LIN {X 0,Y 173.677,Z 475.724,A -85,B 0,C 180,E1 -30232.4,E2 -30232.4} C_VEL
LIN {X 0,Y 173.787,Z 475.712,A -85,B 0,C 180,E1 -30235.65,E2 -30235.65} C_VEL
LIN {X 0,Y 173.897,Z 476.638,A -85,B 0,C 180,E1 -30237.104,E2 -30237.104} C_VEL
LIN {X 0,Y 169.927,Z 506.64,A -85,B 0,C 180,E1 -30237.538,E2 -30237.538} C_VEL
LIN {X 0,Y 166.155,Z 523.912,A -85,B 0,C 180,E1 -30237.792,E2 -30237.792} C_VEL
LIN {X 0,Y 160.855,Z 540.987,A -85,B 0,C 180,E1 -30238.078,E2 -30238.078} C_VEL
LIN {X 0,Y 155.111,Z 555.302,A -85,B 0,C 180,E1 -30238.461,E2 -30238.461} C_VEL
LIN {X 0,Y 147.609,Z 570.627,A -85,B 0,C 180,E1 -30239.029,E2 -30239.029} C_VEL
LIN {X 0,Y 139.67,Z 584.169,A -85,B 0,C 180,E1 -30239.669,E2 -30239.669} C_VEL
LIN {X 0,Y 130.9,Z 596.782,A -85,B 0,C 180,E1 -30240.433,E2 -30240.433} C_VEL
LIN {X 0,Y 121.274,Z 608.767,A -85,B 0,C 180,E1 -30241.51,E2 -30241.51} C_VEL
LIN {X 0,Y 110.826,Z 620.073,A -85,B 0,C 180,E1 -30242.83,E2 -30242.83} C_VEL
LIN {X 0,Y 98.738,Z 631.287,A -85,B 0,C 180,E1 -30244.804,E2 -30244.804} C_VEL
LIN {X 0,Y 86.785,Z 640.843,A -85,B 0,C 180,E1 -30247.242,E2 -30247.242} C_VEL
LIN {X 0,Y 72.974,Z 650.367,A -85,B 0,C 180,E1 -30251.102,E2 -30251.102} C_VEL
LIN {X 0,Y 62.022,Z 656.96,A -85,B 0,C 180,E1 -30255.6,E2 -30255.6} C_VEL
LIN {X 0,Y 49.708,Z 663.438,A -85,B 0,C 180,E1 -30263.221,E2 -30263.221} C_VEL
LIN {X 0,Y 38.747,Z 668.721,A -85,B 0,C 180,E1 -30275.294,E2 -30275.294} C_VEL
LIN {X 0,Y 32.128,Z 671.865,A -85,B 0,C 180,E1 -30288.988,E2 -30288.988} C_VEL
LIN {X 0,Y 27.268,Z 675.138,A -85,B 0,C 180,E1 -30315.066,E2 -30315.066} C_VEL
LIN {X 0,Y 27.051,Z 676.337,A -85,B 0,C 180,E1 -30330.002,E2 -30330.002} C_VEL
LIN {X 0,Y 29.084,Z 677.949,A -85,B 0,C 180,E1 -30358.903,E2 -30358.903} C_VEL
LIN {X 0,Y 36.518,Z 678.543,A -85,B 0,C 180,E1 -30380.339,E2 -30380.339} C_VEL
LIN {X 0,Y 47.081,Z 678.294,A -85,B 0,C 180,E1 -30393.595,E2 -30393.595} C_VEL
LIN {X 0,Y 59.202,Z 677.038,A -85,B 0,C 180,E1 -30401.751,E2 -30401.751} C_VEL
LIN {X 0,Y 72.097,Z 674.944,A -85,B 0,C 180,E1 -30407.114,E2 -30407.114} C_VEL
LIN {X 0,Y 85.435,Z 671.806,A -85,B 0,C 180,E1 -30410.805,E2 -30410.805} C_VEL
LIN {X 0,Y 99.04,Z 667.758,A -85,B 0,C 180,E1 -30413.447,E2 -30413.447} C_VEL
LIN {X 0,Y 103.79,Z 666.021,A -85,B 0,C 180,E1 -30414.851,E2 -30414.851} C_VEL
LIN {X 0,Y 91.479,Z 669.945,A -85,B 0,C 180,E1 -30417.138,E2 -30417.138} C_VEL
LIN {X 0,Y 77.315,Z 673.389,A -85,B 0,C 180,E1 -30420.727,E2 -30420.727} C_VEL
LIN {X 0,Y 71.22,Z 674.56,A -85,B 0,C 180,E1 -30422.724,E2 -30422.724} C_VEL
LIN {X 0,Y 65.681,Z 675.514,A -85,B 0,C 180,E1 -30424.238,E2 -30424.238} C_VEL
LIN {X 0,Y 55.954,Z 676.725,A -85,B 0,C 180,E1 -30425.652,E2 -30425.652} C_VEL
LIN {X 0,Y 48.115,Z 677.331,A -85,B 0,C 180,E1 -30427.013,E2 -30427.013} C_VEL
LIN {X 0,Y 42.491,Z 677.574,A -85,B 0,C 180,E1 -30429.349,E2 -30429.349} C_VEL
LIN {X 0,Y 40.74,Z 677.594,A -85,B 0,C 180,E1 -30430.605,E2 -30430.605} C_VEL
LIN {X 0,Y 30.463,Z 677.43,A -85,B 0,C 180,E1 -30442.652,E2 -30442.652} C_VEL
LIN {X 0,Y 21.513,Z 676.237,A -85,B 0,C 180,E1 -30469.201,E2 -30469.201} C_VEL
LIN {X 0,Y 19.772,Z 674.131,A -85,B 0,C 180,E1 -30509.998,E2 -30509.998} C_VEL
LIN {X 0,Y 22.377,Z 672.647,A -85,B 0,C 180,E1 -30528.302,E2 -30528.302} C_VEL
LIN {X 0,Y 30.887,Z 669.037,A -85,B 0,C 180,E1 -30553.047,E2 -30553.047} C_VEL
LIN {X 0,Y 42.253,Z 664.389,A -85,B 0,C 180,E1 -30566.267,E2 -30566.267} C_VEL
LIN {X 0,Y 54.745,Z 658.555,A -85,B 0,C 180,E1 -30573.978,E2 -30573.978} C_VEL
LIN {X 0,Y 69.55,Z 650.497,A -85,B 0,C 180,E1 -30579.179,E2 -30579.179} C_VEL
LIN {X 0,Y 82.959,Z 641.846,A -85,B 0,C 180,E1 -30582.373,E2 -30582.373} C_VEL
LIN {X 0,Y 96.529,Z 631.523,A -85,B 0,C 180,E1 -30584.728,E2 -30584.728} C_VEL
LIN {X 0,Y 108.467,Z 620.802,A -85,B 0,C 180,E1 -30586.385,E2 -30586.385} C_VEL
LIN {X 0,Y 120.445,Z 608.24,A -85,B 0,C 180,E1 -30587.785,E2 -30587.785} C_VEL
LIN {X 0,Y 130.752,Z 595.563,A -85,B 0,C 180,E1 -30588.796,E2 -30588.796} C_VEL
LIN {X 0,Y 140.255,Z 581.848,A -85,B 0,C 180,E1 -30589.54,E2 -30589.54} C_VEL
LIN {X 0,Y 148.859,Z 566.964,A -85,B 0,C 180,E1 -30590.251,E2 -30590.251} C_VEL
LIN {X 0,Y 155.772,Z 552.366,A -85,B 0,C 180,E1 -30590.729,E2 -30590.729} C_VEL
LIN {X 0,Y 161.828,Z 536.527,A -85,B 0,C 180,E1 -30591.117,E2 -30591.117} C_VEL
LIN {X 0,Y 166.651,Z 520.038,A -85,B 0,C 180,E1 -30591.425,E2 -30591.425} C_VEL
LIN {X 0,Y 170.074,Z 503.577,A -85,B 0,C 180,E1 -30591.604,E2 -30591.604} C_VEL
LIN {X 0,Y 172.803,Z 482.985,A -85,B 0,C 180,E1 -30591.856,E2 -30591.856} C_VEL
LIN {X 0,Y 172.823,Z 482.635,A -85,B 0,C 180,E1 -30594.421,E2 -30594.421} C_VEL
LIN {X 0,Y 172.849,Z 482.63,A -85,B 0,C 180,E1 -30594.821,E2 -30594.821} C_VEL
LIN {X 0,Y 169.394,Z 507.485,A -85,B 0,C 180,E1 -30595.166,E2 -30595.166} C_VEL
LIN {X 0,Y 165.595,Z 524.402,A -85,B 0,C 180,E1 -30595.346,E2 -30595.346} C_VEL
LIN {X 0,Y 160.37,Z 541.058,A -85,B 0,C 180,E1 -30595.551,E2 -30595.551} C_VEL
LIN {X 0,Y 154.582,Z 555.32,A -85,B 0,C 180,E1 -30595.847,E2 -30595.847} C_VEL
LIN {X 0,Y 147.02,Z 570.594,A -85,B 0,C 180,E1 -30596.273,E2 -30596.273} C_VEL
LIN {X 0,Y 138.847,Z 584.351,A -85,B 0,C 180,E1 -30596.773,E2 -30596.773} C_VEL
LIN {X 0,Y 131.044,Z 595.51,A -85,B 0,C 180,E1 -30597.276,E2 -30597.276} C_VEL
LIN {X 0,Y 121.299,Z 607.674,A -85,B 0,C 180,E1 -30598.101,E2 -30598.101} C_VEL
LIN {X 0,Y 110.705,Z 619.069,A -85,B 0,C 180,E1 -30599.075,E2 -30599.075} C_VEL
LIN {X 0,Y 98.397,Z 630.403,A -85,B 0,C 180,E1 -30600.598,E2 -30600.598} C_VEL
LIN {X 0,Y 86.171,Z 640.073,A -85,B 0,C 180,E1 -30602.453,E2 -30602.453} C_VEL
LIN {X 0,Y 74.063,Z 648.403,A -85,B 0,C 180,E1 -30604.926,E2 -30604.926} C_VEL
LIN {X 0,Y 60.474,Z 656.337,A -85,B 0,C 180,E1 -30608.955,E2 -30608.955} C_VEL
LIN {X 0,Y 47.324,Z 662.904,A -85,B 0,C 180,E1 -30615.141,E2 -30615.141} C_VEL
LIN {X 0,Y 35.077,Z 668.267,A -85,B 0,C 180,E1 -30625.632,E2 -30625.632} C_VEL
LIN {X 0,Y 22.994,Z 673.278,A -85,B 0,C 180,E1 -30652.319,E2 -30652.319} C_VEL
LIN {X 0,Y 19.941,Z 676.004,A -85,B 0,C 180,E1 -30690.002,E2 -30690.002} C_VEL
LIN {X 0,Y 23.073,Z 677.681,A -85,B 0,C 180,E1 -30727.534,E2 -30727.534} C_VEL
LIN {X 0,Y 32.417,Z 678.315,A -85,B 0,C 180,E1 -30750.136,E2 -30750.136} C_VEL
LIN {X 0,Y 44.352,Z 678.112,A -85,B 0,C 180,E1 -30761.947,E2 -30761.947} C_VEL
LIN {X 0,Y 57.357,Z 676.918,A -85,B 0,C 180,E1 -30768.599,E2 -30768.599} C_VEL
LIN {X 0,Y 70.839,Z 674.861,A -85,B 0,C 180,E1 -30772.804,E2 -30772.804} C_VEL
LIN {X 0,Y 77.687,Z 673.437,A -85,B 0,C 180,E1 -30774.345,E2 -30774.345} C_VEL
LIN {X 0,Y 78.746,Z 673.197,A -85,B 0,C 180,E1 -30774.882,E2 -30774.882} C_VEL
LIN {X 0,Y 63.264,Z 675.916,A -85,B 0,C 180,E1 -30778.939,E2 -30778.939} C_VEL
LIN {X 0,Y 49.37,Z 677.255,A -85,B 0,C 180,E1 -30784.795,E2 -30784.795} C_VEL
LIN {X 0,Y 40.74,Z 677.594,A -85,B 0,C 180,E1 -30790.605,E2 -30790.605} C_VEL
LIN {X 0,Y 35.42,Z 677.641,A -85,B 0,C 180,E1 -30794.476,E2 -30794.476} C_VEL
LIN {X 0,Y 26.085,Z 677.341,A -85,B 0,C 180,E1 -30800.759,E2 -30800.759} C_VEL
LIN {X 0,Y 18.851,Z 676.794,A -85,B 0,C 180,E1 -30809.438,E2 -30809.438} C_VEL
LIN {X 0,Y 14.47,Z 676.118,A -85,B 0,C 180,E1 -30823.323,E2 -30823.323} C_VEL
LIN {X 0,Y 13.482,Z 675.856,A -85,B 0,C 180,E1 -30830.336,E2 -30830.336} C_VEL
LIN {X 0,Y 12.504,Z 674.478,A -85,B 0,C 180,E1 -30869.996,E2 -30869.996} C_VEL
LIN {X 0,Y 15.718,Z 673.028,A -85,B 0,C 180,E1 -30896.556,E2 -30896.556} C_VEL
LIN {X 0,Y 26.146,Z 669.493,A -85,B 0,C 180,E1 -30923.743,E2 -30923.743} C_VEL
LIN {X 0,Y 38.768,Z 664.885,A -85,B 0,C 180,E1 -30935.011,E2 -30935.011} C_VEL
LIN {X 0,Y 52.028,Z 659.137,A -85,B 0,C 180,E1 -30941.005,E2 -30941.005} C_VEL
LIN {X 0,Y 67.36,Z 651.171,A -85,B 0,C 180,E1 -30944.815,E2 -30944.815} C_VEL
LIN {X 0,Y 81.098,Z 642.622,A -85,B 0,C 180,E1 -30947.142,E2 -30947.142} C_VEL
LIN {X 0,Y 94.914,Z 632.362,A -85,B 0,C 180,E1 -30948.842,E2 -30948.842} C_VEL
LIN {X 0,Y 107.024,Z 621.764,A -85,B 0,C 180,E1 -30950.065,E2 -30950.065} C_VEL
LIN {X 0,Y 119.152,Z 609.349,A -85,B 0,C 180,E1 -30951.102,E2 -30951.102} C_VEL
LIN {X 0,Y 129.567,Z 596.855,A -85,B 0,C 180,E1 -30951.855,E2 -30951.855} C_VEL
LIN {X 0,Y 139.154,Z 583.333,A -85,B 0,C 180,E1 -30952.377,E2 -30952.377} C_VEL
LIN {X 0,Y 146.965,Z 570.192,A -85,B 0,C 180,E1 -30952.877,E2 -30952.877} C_VEL
LIN {X 0,Y 148.7,Z 567.063,A -85,B 0,C 180,E1 -30952.987,E2 -30952.987} C_VEL
LIN {X 0,Y 148.565,Z 567.325,A -85,B 0,C 180,E1 -30953.422,E2 -30953.422} C_VEL
LIN {X 0,Y 140.509,Z 581.212,A -85,B 0,C 180,E1 -30953.775,E2 -30953.775} C_VEL
LIN {X 0,Y 131.68,Z 594.109,A -85,B 0,C 180,E1 -30954.118,E2 -30954.118} C_VEL
LIN {X 0,Y 121.754,Z 606.579,A -85,B 0,C 180,E1 -30954.696,E2 -30954.696} C_VEL
LIN {X 0,Y 111.058,Z 618.049,A -85,B 0,C 180,E1 -30955.336,E2 -30955.336} C_VEL
LIN {X 0,Y 98.588,Z 629.517,A -85,B 0,C 180,E1 -30956.383,E2 -30956.383} C_VEL
LIN {X 0,Y 86.166,Z 639.301,A -85,B 0,C 180,E1 -30957.623,E2 -30957.623} C_VEL
LIN {X 0,Y 72.038,Z 648.779,A -85,B 0,C 180,E1 -30959.585,E2 -30959.585} C_VEL
LIN {X 0,Y 56.298,Z 657.547,A -85,B 0,C 180,E1 -30962.96,E2 -30962.96} C_VEL
LIN {X 0,Y 42.572,Z 663.833,A -85,B 0,C 180,E1 -30967.908,E2 -30967.908} C_VEL
LIN {X 0,Y 29.399,Z 668.912,A -85,B 0,C 180,E1 -30977.022,E2 -30977.022} C_VEL
LIN {X 0,Y 17.863,Z 672.872,A -85,B 0,C 180,E1 -30998.108,E2 -30998.108} C_VEL
LIN {X 0,Y 12.818,Z 675.671,A -85,B 0,C 180,E1 -31050.004,E2 -31050.004} C_VEL
LIN {X 0,Y 17.937,Z 677.391,A -85,B 0,C 180,E1 -31101.599,E2 -31101.599} C_VEL
LIN {X 0,Y 29.503,Z 678.087,A -85,B 0,C 180,E1 -31122.343,E2 -31122.343} C_VEL
LIN {X 0,Y 42.676,Z 677.921,A -85,B 0,C 180,E1 -31131.155,E2 -31131.155} C_VEL
LIN {X 0,Y 49.489,Z 677.458,A -85,B 0,C 180,E1 -31133.775,E2 -31133.775} C_VEL
LIN {X 0,Y 52.007,Z 677.25,A -85,B 0,C 180,E1 -31135.144,E2 -31135.144} C_VEL
LIN {X 0,Y 35.184,Z 677.876,A -85,B 0,C 180,E1 -31142.831,E2 -31142.831} C_VEL
LIN {X 0,Y 21.175,Z 677.138,A -85,B 0,C 180,E1 -31159.395,E2 -31159.395} C_VEL
LIN {X 0,Y 13.482,Z 675.856,A -85,B 0,C 180,E1 -31190.336,E2 -31190.336} C_VEL
LIN {X 0,Y 11.495,Z 675.049,A -85,B 0,C 180,E1 -31215.859,E2 -31215.859} C_VEL
LIN {X 0,Y 11.187,Z 674.089,A -85,B 0,C 180,E1 -31245.852,E2 -31245.852} C_VEL
LIN {X 0,Y 17.142,Z 671.651,A -85,B 0,C 180,E1 -31289.082,E2 -31289.082} C_VEL
LIN {X 0,Y 22.157,Z 670.118,A -85,B 0,C 180,E1 -31297.774,E2 -31297.774} C_VEL
LIN {X 0,Y 23.978,Z 669.538,A -85,B 0,C 180,E1 -31299.324,E2 -31299.324} C_VEL
LIN {X 0,Y 39.801,Z 664.103,A -85,B 0,C 180,E1 -31306.207,E2 -31306.207} C_VEL
LIN {X 0,Y 53.657,Z 658.107,A -85,B 0,C 180,E1 -31309.214,E2 -31309.214} C_VEL
LIN {X 0,Y 68.269,Z 650.459,A -85,B 0,C 180,E1 -31311.014,E2 -31311.014} C_VEL
LIN {X 0,Y 81.57,Z 642.176,A -85,B 0,C 180,E1 -31312.233,E2 -31312.233} C_VEL
LIN {X 0,Y 85.062,Z 639.724,A -85,B 0,C 180,E1 -31312.505,E2 -31312.505} C_VEL
LIN {X 0,Y 84.98,Z 639.793,A -85,B 0,C 180,E1 -31312.939,E2 -31312.939} C_VEL
LIN {X 0,Y 70.665,Z 649.146,A -85,B 0,C 180,E1 -31314.008,E2 -31314.008} C_VEL
LIN {X 0,Y 56.389,Z 656.951,A -85,B 0,C 180,E1 -31315.603,E2 -31315.603} C_VEL
LIN {X 0,Y 38.659,Z 664.745,A -85,B 0,C 180,E1 -31319.015,E2 -31319.015} C_VEL
LIN {X 0,Y 21.257,Z 670.632,A -85,B 0,C 180,E1 -31327.322,E2 -31327.322} C_VEL
LIN {X 0,Y 8.546,Z 674.023,A -85,B 0,C 180,E1 -31354.691,E2 -31354.691} C_VEL
LIN {X 0,Y 5.689,Z 675.338,A -85,B 0,C 180,E1 -31410.008,E2 -31410.008} C_VEL
LIN {X 0,Y 8.613,Z 676.359,A -85,B 0,C 180,E1 -31464.698,E2 -31464.698} C_VEL
LIN {X 0,Y 21.28,Z 677.575,A -85,B 0,C 180,E1 -31492.241,E2 -31492.241} C_VEL
LIN {X 0,Y 24.101,Z 677.729,A -85,B 0,C 180,E1 -31495.561,E2 -31495.561} C_VEL
LIN {X 0,Y 14.131,Z 676.865,A -85,B 0,C 180,E1 -31505.88,E2 -31505.88} C_VEL
LIN {X 0,Y 5.226,Z 674.824,A -85,B 0,C 180,E1 -31589.991,E2 -31589.991} C_VEL
LIN {X 0,Y 10.692,Z 673.192,A -85,B 0,C 180,E1 -31638.878,E2 -31638.878} C_VEL
LIN {X 0,Y 23.978,Z 669.538,A -85,B 0,C 180,E1 -31659.324,E2 -31659.324} C_VEL
LIN {X 0,Y 23.978,Z 669.538,A -85,B 0,C 180,E1 -31659.324,E2 -31659.324}

QRS_NEXT_CUT()

QRS_NEXT()
QRS_HOME()

END
